INTERFACE I_MotionAxisCommonDS402

PROPERTY DS402HomeAborted : BOOL
GET
END_GET
END_PROPERTY

PROPERTY DS402HomeBusy : BOOL
GET
END_GET
END_PROPERTY

PROPERTY DS402HomeDone : BOOL
GET
END_GET
END_PROPERTY

PROPERTY DS402HomeError : BOOL
GET
END_GET
END_PROPERTY

PROPERTY DS402HomeErrorID : UDINT
GET
END_GET
END_PROPERTY

METHOD INTERNAL HomeDS402
VAR_INPUT
    Start: BOOL;
    HomingMethod : E_DS402HomingMethod;
    HomingSpeedsFast : LREAL;
    HomingSpeedsSlow : LREAL;
    HomingAcceleration : LREAL;
    HomeOffset : LREAL;
    UserAbort : BOOL;
    MostRecentModeOfOperation : E_DS402OpMode;
END_VAR
END_METHOD

METHOD SetModeOfOperation : BOOL
VAR_INPUT
    ModeOfOperation : E_DS402OpMode;
END_VAR
END_METHOD

END_INTERFACE

(* stored: Version 1.1.0.1
   Itf I_MotionAxisCommonDS402: Id {5cfa6b6b-bfba-4af4-97dd-dc8ae67741ad}
   Property DS402HomeAborted: Id {a5e8251b-8089-4eac-a5a9-25ef9a79ca2a}
   Get Get: Id {29a04c4d-e661-4810-b596-8fcc9fb61967}
   Property DS402HomeBusy: Id {1b03ac00-4c91-44a8-985f-09513447653c}
   Get Get: Id {0139e914-1b93-4b95-9924-c6f893d4fd03}
   Property DS402HomeDone: Id {ff764d12-550d-4062-920c-53aa0168080e}
   Get Get: Id {cccc1c17-8596-4be0-b798-a92a394e274d}
   Property DS402HomeError: Id {7046f16c-43d0-4904-8195-d98411855d6e}
   Get Get: Id {2fc129d6-09f6-4711-b79c-76dd0df352c1}
   Property DS402HomeErrorID: Id {9c2cad2c-db52-428e-b7bb-6a5288d3b41c}
   Get Get: Id {d46b827f-dbbd-4e59-a309-586db4fec787}
   Method HomeDS402: Id {151ad2ee-1947-4db0-a86f-ef1c83f9e99b}
   Method SetModeOfOperation: Id {0451dd2e-b000-4bfd-b0c5-aec2705c2ae9} *)
